Staubli VAL3: KillAlltasks.pgx

program KillAllTasks()
begin
//*******************************************************************************
//*   ______
//*  / _____) /|
//* | |      / /
//* | | /\  / /
//* | | \ \/ /  _      Copyright (c) KEOLABS, 2016
//* | |  \__/  | |        http://www.keolabs.com
//* | |________| |
//*  \__________/
//*
//********************************************************************************
//*@file          : KillTasks
//*@author        : Yves Ragot
//*@version       : $Id: KillAlltasks.pgx 1191 2016-10-05 15:10:08Z yves $
//*@brief         : kill all running tasks
//*
//*******************************************************************************/

  if taskStatus("COM") != -1
    taskKill("COM")
    wait(taskStatus("COM") == -1)
  endIf

  if taskStatus("Motion") != -1
    taskKill("Motion")
    wait(taskStatus("Motion") == -1)
  endIf

  if taskStatus("CheckStatus") != -1
    taskKill("CheckStatus")
    wait(taskStatus("CheckStatus") == -1)
  endIf

  if taskStatus("CheckLimits") != -1
    taskKill("CheckLimits")
    wait(taskStatus("CheckLimits") == -1)
  endIf

end
